{attribute 'qualified_only'}
{attribute 'strict'}
TYPE E_MA_ROTATOR_TYPE :
(
	DROT 	:= 0,	// Derotator
	ADAPTER := 1,	// Adapter
	ROTATOR := 2	// Rotator
);
END_TYPE

(* stored: Version 1.1.0.1, ProductVersion 3.1.4022.16
   DUT E_MA_ROTATOR_TYPE: Id {3d0c2e7d-59f2-41ff-8db5-5cdde5a63f5d} *)
